// TIA Portal project "Projektet 2.sem" (V16)

(* hardware
DEVICE "S71500/ET200MP station_1"  S7-1500 station
   slot 0: "Rail_0"  Rack  6ES7 590-1***0-0AA0
   slot 1: "PLC_1"  CPU 1516-3 PN/DP  6ES7 516-3AN01-0AB0  V2.0
      slot 3: "CPU display_1"  6ES7591-1BA00-0AA0
      slot 32768: "PROFINET interface_1"  X1
         slot 32769: "Port_1"  X1 P1
         slot 32770: "Port_2"  X1 P2
      slot 33024: "PROFINET interface_2"  X2
         slot 33025: "Port_1"  X2 P1
      slot 33280: "DP interface_1"  X3
   slot 2: "DI 32x24VDC HF_1"  DI 32x24VDC HF  6ES7 521-1BL00-0AB0  V2.0
   slot 3: "DQ 32x24VDC/0.5A HF_1"  DQ 32x24VDC/0.5A HF  6ES7 522-1BL01-0AB0  V1.0
   slot 4: "AI 8xU/I/RTD/TC ST_1"  AI 8xU/I/RTD/TC ST  6ES7 531-7KF00-0AB0  V2.0
   slot 5: "AQ 4xU/I ST_1"  AQ 4xU/I ST  6ES7 532-5HD00-0AB0  V2.0
DEVICE "HMI_1"  KTP700 Basic PN
   slot 0: "HMI_1"  KTP700 Basic PN  6AV2 123-2GB03-0AX0  16.0.0.0
   slot 1: "HMI_RT_1"  KTP700 Basic PN  6AV2 123-2GB03-0AX0  16.0.0.0
   slot 5: "HMI_1.IE_CP_1"  PROFINET Interface  16.0.0.0
      slot 1: "PROFINET Interface_1"  PROFINET Interface
         slot 1: "Port_1"  Port
*)

// ===== PLC "PLC_1"  CPU 1516-3 PN/DP =====

VAR_GLOBAL   // PLC tag table "Default tag table"
   "FMA-B1" AT %I0.0 : Bool;
   "FMA-B2" AT %I0.1 : Bool;
   "FMA-B3" AT %I0.2 : Bool;
   "FMA-M1f" AT %Q0.0 : Bool;
   "FMA-M1r" AT %Q0.1 : Bool;
   "FMA-M2" AT %Q0.2 : Bool;
   "FMB-B1" AT %I100.0 : Bool;
   "FMB-B2" AT %I100.1 : Bool;
   "FMB-B3" AT %I100.2 : Bool;
   "FMB-B4" AT %I100.3 : Bool;
   "FMB-B5" AT %I100.4 : Bool;
   "FMB-B6" AT %I100.5 : Bool;
   "FMB-M1" AT %Q100.0 : Bool;
   "FMB-M2" AT %Q100.1 : Bool;
   "FMB-M3" AT %Q100.2 : Bool;
   "FMB-M4" AT %Q100.3 : Bool;
   "Start/reset" AT %M5.0 : Bool;
   "Aktuel sekvens" AT %MW20 : Int;
   "EmneIsFaulty" AT %M5.1 : Bool;
   "ID" AT %MW22 : Int;
   "counter" AT %MW24 : Int;
   "RunOneTime" AT %M5.2 : Bool;
   "RunOneTime(1)" AT %M5.3 : Bool;
   "Test" AT %M2.0 : Bool;
   "Test(1)" AT %M2.1 : Bool;
   "System_Byte" AT %MB1 : Byte;
   "FirstScan" AT %M1.0 : Bool;
   "DiagStatusUpdate" AT %M1.1 : Bool;
   "AlwaysTRUE" AT %M1.2 : Bool;
   "AlwaysFALSE" AT %M1.3 : Bool;
   "Clock_Byte" AT %MB0 : Byte;
   "Clock_10Hz" AT %M0.0 : Bool;
   "Clock_5Hz" AT %M0.1 : Bool;
   "Clock_2.5Hz" AT %M0.2 : Bool;
   "Clock_2Hz" AT %M0.3 : Bool;
   "Clock_1.25Hz" AT %M0.4 : Bool;
   "Clock_1Hz" AT %M0.5 : Bool;
   "Clock_0.625Hz" AT %M0.6 : Bool;
   "Clock_0.5Hz" AT %M0.7 : Bool;
END_VAR

DATA_BLOCK "Database"   // DB1
{ S7_Optimized_Access := 'FALSE' }
VERSION : 0.1
   VAR
      Queue : Array[0..19] of Int;
      Finished : Array[0..1999] of Int;
      Status : Array[0..1999] of Bool;
   END_VAR
BEGIN
END_DATA_BLOCK

// folder: System blocks/Program resources

DATA_BLOCK "IEC_Timer_0_DB"   // DB2
{ S7_Optimized_Access := 'TRUE' }
AUTHOR : Simatic
FAMILY : IEC
NAME : IEC_TMR
VERSION : 1.0
// stored: InstanceOfName IEC_TIMER
"IEC_TIMER"
BEGIN
END_DATA_BLOCK

// folder: (top level)

FUNCTION "Sekvens" : Void   // FC1, LAD
{ S7_Optimized_Access := 'TRUE' }
VERSION : 0.1
   VAR_TEMP   // added for the SCL form of the ladder/FBD networks
      _w1 : Bool;
   END_VAR
BEGIN

REGION Network 1
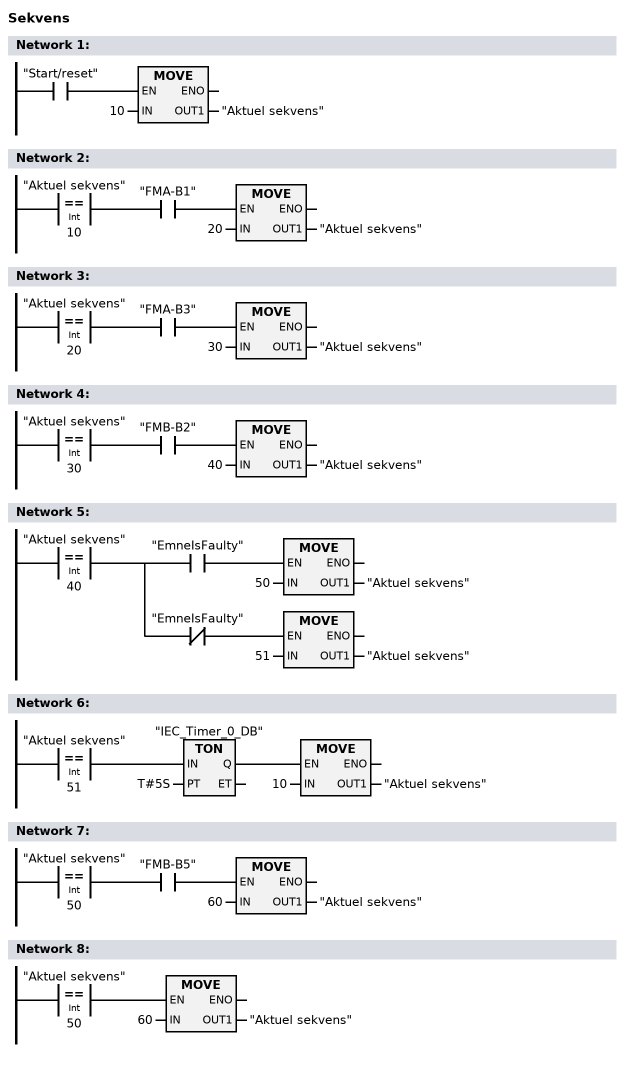
   RUNG wire#powerrail
      Contact( "Start/reset" )
      Move(in := 10, out1 => "Aktuel sekvens")
   END_RUNG
   // the same network as SCL:
   IF "Start/reset" THEN "Aktuel sekvens" := 10; END_IF;
END_REGION

REGION Network 2
   RUNG wire#powerrail
      { S7_Templates := "SrcType := Int" } EQ_Contact(in1 := "Aktuel sekvens", in2 := 10)
      Contact( "FMA-B1" )
      Move(in := 20, out1 => "Aktuel sekvens")
   END_RUNG
   // the same network as SCL:
   IF ("Aktuel sekvens" = 10) AND "FMA-B1" THEN "Aktuel sekvens" := 20; END_IF;
END_REGION

REGION Network 3
   RUNG wire#powerrail
      { S7_Templates := "SrcType := Int" } EQ_Contact(in1 := "Aktuel sekvens", in2 := 20)
      Contact( "FMA-B3" )
      Move(in := 30, out1 => "Aktuel sekvens")
   END_RUNG
   // the same network as SCL:
   IF ("Aktuel sekvens" = 20) AND "FMA-B3" THEN "Aktuel sekvens" := 30; END_IF;
END_REGION

REGION Network 4
   RUNG wire#powerrail
      { S7_Templates := "SrcType := Int" } EQ_Contact(in1 := "Aktuel sekvens", in2 := 30)
      Contact( "FMB-B2" )
      Move(in := 40, out1 => "Aktuel sekvens")
   END_RUNG
   // the same network as SCL:
   IF ("Aktuel sekvens" = 30) AND "FMB-B2" THEN "Aktuel sekvens" := 40; END_IF;
END_REGION

REGION Network 5
   RUNG wire#powerrail
      { S7_Templates := "SrcType := Int" } EQ_Contact(in1 := "Aktuel sekvens", in2 := 40)
      wire#w1
      Contact( "EmneIsFaulty" )
      Move(in := 50, out1 => "Aktuel sekvens")
   END_RUNG
   RUNG wire#w1
      I_Contact( "EmneIsFaulty" )
      Move(in := 51, out1 => "Aktuel sekvens")
   END_RUNG
   // the same network as SCL:
   #_w1 := "Aktuel sekvens" = 40;
   IF #_w1 AND "EmneIsFaulty" THEN "Aktuel sekvens" := 50; END_IF;
   IF #_w1 AND NOT "EmneIsFaulty" THEN "Aktuel sekvens" := 51; END_IF;
END_REGION

REGION Network 6
   "IEC_Timer_0_DB".TON(IN := "Aktuel sekvens" = 51, PT := T#5S);
   IF "IEC_Timer_0_DB".Q THEN "Aktuel sekvens" := 10; END_IF;
END_REGION

REGION Network 7
   RUNG wire#powerrail
      { S7_Templates := "SrcType := Int" } EQ_Contact(in1 := "Aktuel sekvens", in2 := 50)
      Contact( "FMB-B5" )
      Move(in := 60, out1 => "Aktuel sekvens")
   END_RUNG
   // the same network as SCL:
   IF ("Aktuel sekvens" = 50) AND "FMB-B5" THEN "Aktuel sekvens" := 60; END_IF;
END_REGION

REGION Network 8
   RUNG wire#powerrail
      { S7_Templates := "SrcType := Int" } EQ_Contact(in1 := "Aktuel sekvens", in2 := 50)
      Move(in := 60, out1 => "Aktuel sekvens")
   END_RUNG
   // the same network as SCL:
   IF "Aktuel sekvens" = 50 THEN "Aktuel sekvens" := 60; END_IF;
END_REGION
END_FUNCTION

FUNCTION "Queue/ID" : Void   // FC2, SCL
{ S7_Optimized_Access := 'TRUE' }
VERSION : 0.1
   VAR_TEMP
      i : Int;
   END_VAR
BEGIN
   //add id to item and put them in queue
   IF "FMA-B1" AND ("RunOneTime" = FALSE) THEN
       "RunOneTime" := TRUE;
       "ID" := "ID" + 1;
       "Database".Finished["ID"] := "ID";
       "Database".Queue["counter"] := "Database".Finished["ID"];
       "counter" := "counter" + 1;
   END_IF;

   //reset function
   IF "RunOneTime" THEN
       IF "FMA-B1" = FALSE THEN
           "RunOneTime" := FALSE;
       END_IF;
   END_IF;
END_FUNCTION

FUNCTION "Check" : Void   // FC3, SCL
{ S7_Optimized_Access := 'TRUE' }
VERSION : 0.1
   VAR_TEMP
      i : Int;
      "Remove from queue" : Bool;
      Retest : Bool;
      temp : Array[0..19] of Int;
   END_VAR
BEGIN
   IF "FMA-B3" THEN
       IF "EmneIsFaulty" AND ("RunOneTime(1)" = FALSE) THEN
           "RunOneTime(1)" := TRUE;
           IF "Database".Status["Database".Queue[0]] THEN
               #"Remove from queue" := TRUE;
           ELSE
               "Database".Status["Database".Queue[0]] := TRUE;
               #Retest := TRUE;
           END_IF;
       ELSIF "RunOneTime(1)" = FALSE THEN
           "Database".Status["Database".Queue[0]] := FALSE;
           #"Remove from queue" := TRUE;
           "RunOneTime(1)" := TRUE;
       END_IF;
   END_IF;


   IF "FMA-B3" = FALSE THEN
       IF "RunOneTime(1)" THEN
           "RunOneTime(1)" := FALSE;
       END_IF;
   END_IF;

   IF #"Remove from queue" THEN
       #"Remove from queue" := FALSE;
       "counter" := "counter" - 1;
       FOR #i := 0 TO 18 DO
           "Database".Queue[#i] := "Database".Queue[#i + 1];
       END_FOR;
   END_IF;

   IF #Retest THEN
       #Retest := FALSE;
       (* "Database".Queue["counter"] := "Database".Queue["counter" - 1];
       "Database".Queue["counter" - 1] := "Database".Queue[0]; *)
       FOR #i := 0 TO 19 DO
           #temp[#i] := "Database".Queue[#i];
       END_FOR;

       FOR #i := 3 TO 19 DO
           "Database".Queue[#i] := #temp[#i - 1];
       END_FOR;
       "Database".Queue[2] := "Database".Queue[0];

       FOR #i := 0 TO 18 DO
           "Database".Queue[#i] := "Database".Queue[#i + 1];
       END_FOR;

   END_IF;
END_FUNCTION

ORGANIZATION_BLOCK "Main"   // OB1, LAD, ProgramCycle
TITLE = "Main Program Sweep (Cycle)"
{ S7_Optimized_Access := 'TRUE' }
VERSION : 0.1
   VAR_INPUT
      Initial_Call : Bool;   // Initial call of this OB
      Remanence : Bool;   // =True, if remanent data are available
   END_VAR
BEGIN

REGION Network 1
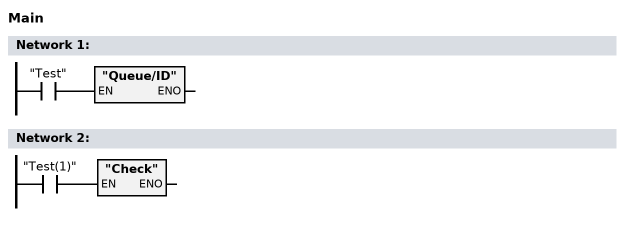
   RUNG wire#powerrail
      Contact( "Test" )
      "Queue/ID"()
   END_RUNG
   // the same network as SCL:
   IF "Test" THEN "Queue/ID"(); END_IF;
END_REGION

REGION Network 2
   RUNG wire#powerrail
      Contact( "Test(1)" )
      "Check"()
   END_RUNG
   // the same network as SCL:
   IF "Test(1)" THEN "Check"(); END_IF;
END_REGION
END_ORGANIZATION_BLOCK

(* ===== HMI "HMI_RT_1" =====
system functions are stored by id; their names below are inferred from use
connection "HMI_Connection_1": ETHERNET, SMART_S7_1500_OMS

HMI tags "Default tag table"
   "Tag_ScreenNumber" : UInt, internal
   "Login_Name" : WString[254], internal
   "Login_Password" : WString[254], internal
   "username" : WString[254], internal

screen "Root screen" 800x480, template "StartSkærm"
   on GenerateScreen: SetTag("Tag_ScreenNumber", 1)
   IOField "I/O field_1" at 317,119 size 175x47; FormatPattern ????????????????????????????????????????????????????????????????????????????????
      ProcessValue <- "Login_Name"
      on Activate: function_a3fbdc78(N)
   IOField "I/O field_2" at 317,198 size 175x47; FormatPattern ????????????????????????????????????????????????????????????????????????????????
      ProcessValue <- "Login_Password"
   TextField "Text field_1" at 197,207 size 115x23; Text 'Adgangskode'
   TextField "Text field_2" at 197,129 size 99x23; Text 'Brugernavn'
   Button "Button_1" at 357,280 size 96x32; TextOff 'Login'
      on Click: function_a9b89908("Login_Password", "Login_Name"); function_f41c6f6c("username")

Template "Tekinker_template" 800x480
   Button "Template_Button_1" at 480,12 size 91x32; TextOff 'Logoff'
      on Click: function_f23ef4c9(); ActivateScreen("Root screen", 0)
   DateTimeField "Template_Date/time field_1" at 578,12 size 219x32
   TextField "Template_Text field_1" at 31,12 size 177x23; Text 'Vaccine Gruppen A/S'
   IOField "Template_I/O field_1" at 291,12 size 181x32; FormatPattern ????????????????????????????????????????????????????????????????????????????????
      ProcessValue <- "username"
   Button "Template_Button_3" at 71,440 size 96x32; TextOff 'I/O Test'; Authorization "Operate"
      on Click: ActivateScreen(N, 0)
   Button "Template_Button_4" at 179,440 size 96x32; TextOff 'UR 3'; Authorization "Operate"
   Button "Template_Button_5" at 287,440 size 96x32; TextOff 'Brugerliste'; Authorization "User administration"
      on Click: ActivateScreen("Brugerliste", 0)
   Button "Template_Button_6" at 502,440 size 96x32; TextOff 'Fejllog'; Authorization "Operate"
      on Click: ActivateScreen("Fejllog", 0)
   Button "Template_Button_7" at 610,440 size 96x32; TextOff 'Tekniker'; Authorization "Operate"
   Button "Template_Button_2" at 394,440 size 96x32; TextOff 'Brugerlog'; Authorization "Operate"
      on Click: ActivateScreen("Brugerlog", 0)
   Button "Template_Button_8" at 610,440 size 96x32; TextOff 'Operatør'; Authorization "Operate"
      on Click: ActivateScreen("Operatør_Skærm", 0)

Template "StartSkærm" 800x480
   DateTimeField "Template_Date/time field_1" at 578,12 size 219x32
   TextField "Template_Text field_1" at 31,12 size 177x23; Text 'Vaccine Gruppen A/S'

screen "Brugerliste" 800x480, template "Tekinker_template"
   UserView "User view_1" at 9,57 size 782x374

screen "Operatør_Skærm" 800x480, template "Operatør_template"
   TextField "Text field_1" at 53,55 size 57x23; Text 'Status'
   TextField "Text field_3" at 178,83 size 69x23; Text 'Fejlrate'
   TextField "Text field_2" at 56,82 size 54x23; Text 'I Drift'
   TextField "Text field_4" at 4,82 size 35x23; Text 'Fejl'
   TextField "Text field_5" at 112,83 size 42x23; Text 'Stop'
   Button "Button_1" at 40,148 size 227x77; TextOff 'Start'; Authorization "Monitor"
   Button "Button_2" at 39,247 size 227x77; TextOff 'Stop'; Authorization "Monitor"
   Button "Button_3" at 38,346 size 227x77; TextOff 'Reset'; Authorization "Monitor"
   TextField "Text field_6" at 447,61 size 195x23; Text 'Information siden login'
   TextField "Text field_7" at 357,97 size 77x23; Text 'Testede:'
   TextField "Text field_8" at 357,134 size 100x23; Text 'Godkendte:'
   TextField "Text field_9" at 357,171 size 58x23; Text 'Fejlet:'
   IOField "I/O field_1" at 513,94 size 96x26; FormatPattern 9999999
   IOField "I/O field_2" at 513,131 size 96x26; FormatPattern 9999999
   IOField "I/O field_3" at 513,168 size 96x26; FormatPattern 9999999
   TextField "Text field_10" at 357,208 size 69x23; Text 'Fejlrate'
   IOField "I/O field_4" at 513,205 size 96x26; FormatPattern 9999999
   TextField "Text field_11" at 412,249 size 323x23; Text 'Information over de sidste 100 testede'
   TextField "Text field_12" at 357,286 size 77x23; Text 'Testede:'
   TextField "Text field_13" at 357,323 size 100x23; Text 'Godkendte:'
   TextField "Text field_14" at 357,360 size 58x23; Text 'Fejlet:'
   IOField "I/O field_5" at 513,283 size 96x28; FormatPattern 9999999
   IOField "I/O field_6" at 513,320 size 96x28; FormatPattern 9999999
   IOField "I/O field_7" at 513,357 size 96x28; FormatPattern 9999999
   TextField "Text field_15" at 357,397 size 69x23; Text 'Fejlrate'
   IOField "I/O field_8" at 513,394 size 96x28; FormatPattern 9999999

screen "Fejllog" 800x480, template "Tekinker_template"
   AlarmView "Alarm view_1" at 8,57 size 787x374; ColumnTextTime 'Tid'; ColumnTextDate 'Dato'; ColumnTextAlarmText 'Log'

screen "Brugerlog" 800x480, template "Tekinker_template"
   AlarmView "Alarm view_1" at 8,57 size 787x374; ColumnTextTime 'Tid'; ColumnTextDate 'Dato'; ColumnTextAlarmText 'Log'
*)